FUNCTION_BLOCK List
VAR_INPUT
END_VAR
VAR_OUTPUT
	count : UINT;
	_typeClass : __SYSTEM.TYPE_CLASS; // Type of data object - primitives or Userdef
	_classSize : DINT; // Size of data object - useful to check type of Userdef typeclass
END_VAR
VAR
	head : POINTER TO Node := NULL;
	tail : POINTER TO Node := NULL;
END_VAR


// linked list implementation reference:
// https://www.codesdope.com/blog/article/c-linked-lists-in-c-singly-linked-list/

(*
	Will try to create list which can contain custom FB as datatype.
	Currently I'm trying to accomplish this using interfaces.

	Maybe this will help
	https://aticleworld.com/generic-linked-list-in-c/
	
	In ListTest/../MAIN are experiments with creation of data


*)


METHOD Append : REFERENCE TO List
VAR_INPUT
	data : ANY;
END_VAR
VAR
	new : POINTER TO Node;
END_VAR

Append REF= THIS^;

IF NOT IsTypeClassCorrect(data) THEN
	RETURN;
END_IF
SetTypeClass(data);

new := __NEW(Node);
new^.data := __NEW(BYTE, classSize);
MEMCPY(new^.data, data.pValue, classSize);
new^.next := NULL;

IF head = NULL THEN
	head := new;
	tail := new;
ELSE
	tail^.next := new;
	tail := tail^.next;
END_IF
count := count + 1;
END_METHOD


//{attribute 'monitoring' := 'call'}
// Size of data object - useful to check type of Userdef typeclass
PROPERTY classSize : DINT
GET

classSize := _classSize;
END_GET
SET // PRIVATE

_classSize := classSize;
END_SET
END_PROPERTY


METHOD FB_init : BOOL
VAR_INPUT
	bInitRetains : BOOL; // if TRUE, the retain variables are initialized (warm start / cold start)
	bInCopyCode : BOOL;  // if TRUE, the instance afterwards gets moved into the copy code (online change)
END_VAR
END_METHOD


METHOD Get : REFERENCE TO List
VAR_INPUT
	// indexing from end allowed
	// index = 0 returns first element
	// index = 1 returns seconds element
	// index = -1 returns last element
	// index = -2 return before-last element
	index : INT;
	destinationVariable : ANY;
END_VAR
VAR
	current : POINTER TO Node := NULL;
	getIndex : INT;
	i : INT;
END_VAR

IF NOT IsTypeClassCorrect(destinationVariable) THEN
	RETURN;
END_IF;

IF head = NULL THEN
	RETURN;
END_IF;

// Calculate actual index in List
getIndex := (count * BOOL_TO_INT(index < 0)) + index;

// Return 0 for invalid indexes
IF 	(getIndex >= count) OR	// Indexing from begin begins with 0
	(getIndex < 0) // Indexing from end begins with -1
THEN
	RETURN;
END_IF


current := head;
FOR i := 1 TO getIndex DO // we already got head in previous line, that's why it's from 1
	IF current^.next = NULL THEN
		RETURN;
	END_IF
	current := current^.next;
END_FOR
MEMMOVE(destinationVariable.pValue, current^.data, classSize);
END_METHOD

// Inserts new element into given index. Negative indexing is supported
METHOD Insert : REFERENCE TO List
VAR_INPUT
	(*
		0 = Prepend;
		1 = Insert into second position;
		-2 = Insert into second position from end;
		-1 = Append;
	*)
	index : INT;
	data : ANY;
END_VAR
VAR
	new : POINTER TO Node;
	current : POINTER TO Node;
	insertIndex : INT;
	i : INT;
END_VAR

Insert REF= THIS^;

IF NOT IsTypeClassCorrect(data) THEN
	RETURN;
END_IF
SetTypeClass(data);

new := __NEW(Node);
new^.data := __NEW(BYTE, classSize);
MEMCPY(new^.data, data.pValue, classSize);

// Calculate actual index in List
insertIndex := ((count + 1) * BOOL_TO_INT(index < 0)) + index;

IF insertIndex >= count // Index too high -> append to end
THEN
	Append(data);
	RETURN;
ELSIF insertIndex <= 0 // Index too high from the end -> prepend to beginning
THEN
	Prepend(data);
	RETURN;
END_IF

current := head;
FOR i := 1 TO insertIndex - 1 DO
	current := current^.next;
END_FOR
new^.next := current^.next;
current^.next := new;
count := count + 1;
END_METHOD


METHOD IsEmpty : BOOL
VAR_INPUT
END_VAR

IsEmpty := head = NULL;
END_METHOD


METHOD IsTypeClassCorrect : BOOL
VAR_INPUT
	CheckedVariable : ANY;
END_VAR

IF classSize = 0 THEN
	IsTypeClassCorrect := TRUE;
	RETURN;
END_IF
IsTypeClassCorrect := typeClass = CheckedVariable.TypeClass AND classSize = CheckedVariable.diSize;
END_METHOD


// Pushes data to the beginning of the list
METHOD Prepend : REFERENCE TO List
VAR_INPUT
	data : ANY;
END_VAR
VAR
	new : POINTER TO Node;
END_VAR

Prepend REF= THIS^;

IF NOT IsTypeClassCorrect(data) THEN
	RETURN;
END_IF
SetTypeClass(data);

new := __NEW(Node);
new^.data := __NEW(BYTE, classSize);
MEMCPY(new^.data, data.pValue, classSize);
new^.next := head;

IF head = NULL THEN
	head := new;
	tail := new;
ELSE
	head := new;
END_IF
count := count + 1;
END_METHOD


METHOD Remove : REFERENCE TO List;
VAR_INPUT
	index : INT;
END_VAR
VAR
	current : POINTER TO Node := NULL;
	removeIndex : INT;	
	nodeToRemove : POINTER TO Node;
	i : INT;
END_VAR

Remove REF= THIS^;

IF head = NULL THEN
	RETURN;
END_IF;

// Calculate actual index in List
removeIndex := (count * BOOL_TO_INT(index < 0)) + index; 

// Cancel removal for invalid indexes
IF 	(removeIndex >= count) OR // Indexing from begin begins with 0
	(removeIndex < 0) // Indexing from end begins with -1
THEN
	RETURN;
END_IF

IF removeIndex = 0 THEN
	nodeToRemove := head;
	head := head^.next;
ELSE
	current := head;
	FOR i := 1 TO removeIndex - 1 DO
		current := current^.next;
	END_FOR
	nodeToRemove := current^.next;
	current^.next := current^.next^.next;
END_IF
IF nodeToRemove = tail THEN
	tail := current;
END_IF
__DELETE(nodeToRemove^.data);
__DELETE(nodeToRemove);
count := count - 1;
END_METHOD


METHOD RemoveAll : REFERENCE TO List
VAR_INPUT
END_VAR

WHILE head <> NULL DO
	Remove(0);
END_WHILE
END_METHOD


METHOD SetTypeClass : BOOL
VAR_INPUT
	ReferenceVariable : ANY; // Pass any variable of your chosen type. It will only be used to obtain data type
END_VAR

IF classSize = 0 THEN
	typeClass := ReferenceVariable.TypeClass;
	classSize := ReferenceVariable.diSize;
	SetTypeClass := TRUE;
END_IF
END_METHOD


//{attribute 'monitoring' := 'call'}
// Type of data object - primitives or Userdef
PROPERTY typeClass : __SYSTEM.TYPE_CLASS
GET

typeClass := _typeClass;
END_GET
SET // PRIVATE

_typeClass := typeClass;
END_SET
END_PROPERTY

END_FUNCTION_BLOCK

(* stored: Version 1.1.0.1, ProductVersion 3.1.4024.11
   POU List: Id {36da1aad-070e-4dc9-a97f-6804d8c29941}, SpecialFunc None
   Method Append: Id {1e1f09ec-b8ab-4564-bd5e-1ec5942968a2}
   Property classSize: Id {7e6085c6-96ce-42a1-8b88-7186e2707c52}
   Get Get: Id {751ed563-245e-4251-8f48-793bea02d2dd}
   Set Set: Id {d28883e4-09ef-4987-9ae9-de437f5febd2}
   Method FB_init: Id {0226c1a8-7221-49d2-9651-621473e3dd48}
   Method Get: Id {27f0a3aa-73ee-439b-a440-9d7ae0b874e3}
   Method Insert: Id {c7ac0742-b796-46ea-b82a-ea65ec86bf7a}
   Method IsEmpty: Id {48c36a62-7159-4bac-9043-c9f34faa0784}
   Method IsTypeClassCorrect: Id {a44011b5-3af2-40fa-9e34-3ea3daf7471f}
   Method Prepend: Id {4d27f5a1-2c00-46ed-9bca-6cb1700691e9}
   Method Remove: Id {a48b451e-3e6f-4bbb-a1ce-018cff54d99b}
   Method RemoveAll: Id {76f34ed4-1c4a-47a9-9afe-52cf0b0c1d2d}
   Method SetTypeClass: Id {f5a2b55d-ed3e-4b78-b26b-e15a7ca8b768}
   Property typeClass: Id {5edcf55a-3211-4d79-ad6d-72dde1f06a69}
   Get Get: Id {338c0731-2dbe-41a5-a853-32e34c8bf6c9}
   Set Set: Id {78ff5002-68b7-404a-bc4f-5a51efac81b5} *)
